{attribute 'linkalways'} 
{attribute 'no_explicit_call' := 'This FB is a CLASS and must be accessed using methods or properties'}
{attribute 'enable_dynamic_creation'}
FUNCTION_BLOCK FINAL XOR_SINT EXTENDS Node
VAR
	in1 : _SINT(0);
	in2 : _SINT(0);
	out : _SINT(0);
END_VAR

METHOD PUBLIC Clone : I_Node
VAR
	pNode : POINTER TO XOR_SINT;
END_VAR
pNode := __NEW(XOR_SINT);
Clone := pNode^;
END_METHOD

METHOD FB_init : BOOL
VAR_INPUT
	bInitRetains : BOOL; // if TRUE, the retain variables are initialized (warm start / cold start)
	bInCopyCode : BOOL;  // if TRUE, the instance afterwards gets moved into the copy code (online change)
END_VAR
AddInput('in1',THIS^.in1);
AddInput('in2',THIS^.in2);
AddOutput('out', THIS^.out);
END_METHOD

METHOD PROTECTED OnExecute
VAR
END_VAR
out.Value := in1.Value XOR in2.Value;
END_METHOD

END_FUNCTION_BLOCK

(* stored: Version 1.1.0.1, ProductVersion 3.1.4024.15
   POU XOR_SINT: Id {0afab56e-e103-468a-92e9-eb5d924e7910}, SpecialFunc None
   Folder Constructor: Id {09183451-39cf-400d-9c2f-b505e5568eea}
   Method Clone: Id {cb5f568d-bc6e-432d-ae77-19b4da89a561}
   Method FB_init: Id {be24cd50-8421-49b0-9858-2a36a47aeb67}
   Method OnExecute: Id {dd7da47e-c187-443e-a339-42212cd95134} *)
